// SIMATIC S7-200 SMART project (STEP 7-Micro/WIN SMART), CPU ST40

SYMBOL_TABLE 系统符号
Always_On        SM0.0    // 始终接通
END_SYMBOL_TABLE

ORGANIZATION_BLOCK MAIN:OB1
TITLE=程序注释
BEGIN
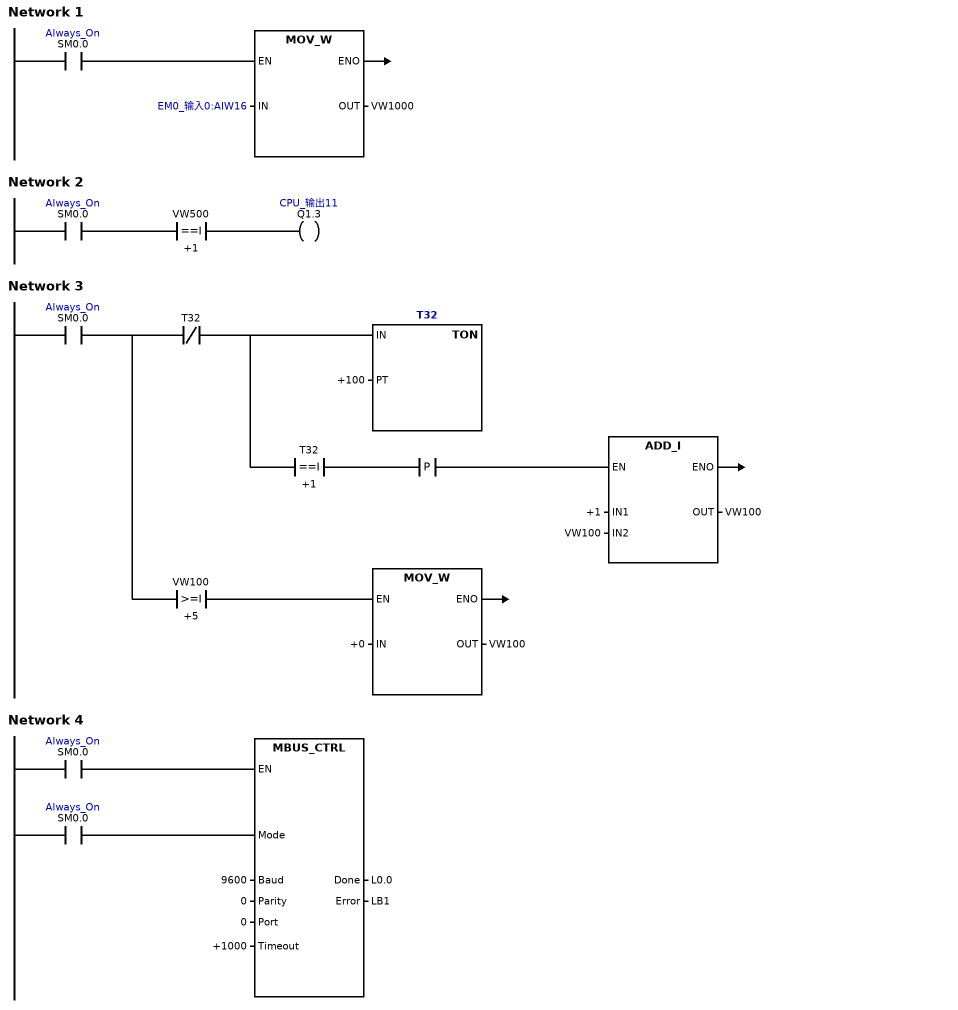
Network 1
LD     Always_On:SM0.0
MOVW   EM0_输入0:AIW16, VW1000
Network 2
LD     Always_On:SM0.0
AW=    VW500, +1
=      CPU_输出11:Q1.3
Network 3
LD     Always_On:SM0.0
LPS
AN     T32
TON    T32, +100
AW=    T32, +1
EU
+I     +1, VW100
LPP
AW>=   VW100, +5
MOVW   +0, VW100
Network 4
LD     Always_On:SM0.0
=      L60.0
LD     Always_On:SM0.0
=      L63.7
LD     L60.0
CALL   MBUS_CTRL:SBR5, L63.7, 9600, 0, 0, +1000, L0.0, LB1
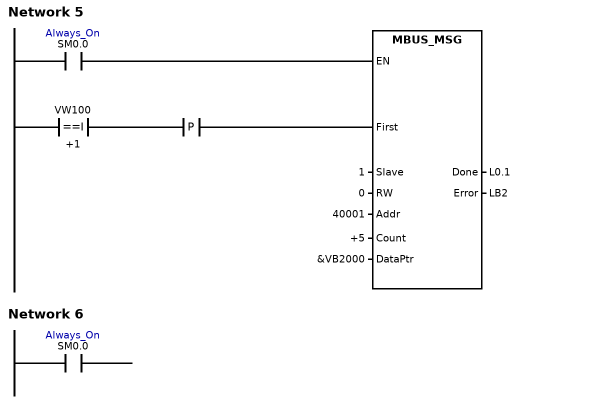
Network 5
LD     Always_On:SM0.0
=      L60.0
LDW=   VW100, +1
EU
=      L63.7
LD     L60.0
CALL   MBUS_MSG:SBR6, L63.7, 1, 0, 40001, +5, &VB2000, L0.1, LB2
Network 6
// (network saved uncompiled; LAD cells follow)
// row 0: c0 -| |- Always_On:SM0.0
END_ORGANIZATION_BLOCK

// SBR1: protected block, not included

// SBR2: protected block, not included

// SBR3: protected block, not included

// SBR4: protected block, not included

// SBR5: protected block, not included

// SBR6: protected block, not included

// SBR7: protected block, not included

// INT1: protected block, not included
